// TIA Portal V20 export
// export: Created 2025-12-01T14:57:45.3823092Z, ExportSetting None, DisplayName Totally Integrated Automation Portal, DisplayVersion V20 Update 3, DisplayName TIA Portal Openness, DisplayVersion V20 Update 3, DisplayName TIA Portal Version Control Interface, DisplayVersion V20 Update 3, DisplayName STEP 7 Professional, DisplayVersion V20 Update 3, DisplayName STEP 7 Safety, DisplayVersion V20 Update 2, DisplayName WinCC Basic/Comfort/Advanced, DisplayVersion V20 Update 3, DisplayName WinCC Professional, DisplayVersion V20 Update 3, DisplayName WinCC Unified, DisplayVersion V20 Update 3
FUNCTION "FC818_Mensaje_BBDD_Routing_Llena" : Void   // FC818, LAD
{ S7_Optimized_Access := 'FALSE' }
// stored: AutoNumber false, SetENOAutomatically false
   VAR_INPUT
      Etiqueta : ULInt;
      Envio_JDT2 : Bool;
   END_VAR
   VAR_TEMP
      Guardar_AR1 : DWord;
      DBEventos : Word;   // Numero del DB de Eventos
      PunteroEventos : DWord;   // Puntero al DB de Eventos
      MaxBytes : UInt;
      NDB_Eventos_Emi : UInt;
      NumBytes : UInt;   // Numero de Bytes existentes en el DB de Eventos
      etiqueta_string : String;
      indice : Int;
      longitud : Int;
      posicion : Int;
      i : Int;
      codigo_string : String[20];
   END_VAR
BEGIN

REGION Network 1 (SCL)
   // buscamos hueco en el db donde vamos a escribir los eventos antes de empezar la conversión
   // 


   IF #Envio_JDT2    = true THEN
       REGION buscar en JDT2

           #posicion := -1;
           FOR #i := 0 TO 100 BY 1 DO
               #longitud := LEN("DB197_eventos_generados_routing_JDT2".evento[#i]);
               IF #longitud = 0 THEN
                   #posicion := #i;
                   EXIT;
               END_IF;
           END_FOR;

           // si no hay sitio para escribir salimos del bloque
           IF #posicion = -1 THEN
               RETURN;
           END_IF;
       END_REGION
       ;
   ELSE
       REGION buscar en JDT1

           #posicion := -1;
           FOR #i := 0 TO 100 BY 1 DO
               #longitud := LEN("DB198_eventos_generados_routing_JDT1".evento[#i]);
               IF #longitud = 0 THEN
                   #posicion := #i;
                   EXIT;
               END_IF;
           END_FOR;

           // si no hay sitio para escribir salimos del bloque
           IF #posicion = -1 THEN
               RETURN;
           END_IF;
       END_REGION
   END_IF;
END_REGION

REGION Network 2 (SCL): formatear el evento


   #codigo_string := DELETE(IN := (ULINT_TO_STRING(IN := #Etiqueta)), L := 1, P := 1);
   // concatenamos el mensaje 
   // 
   IF #Envio_JDT2= true THEN

       "DB197_eventos_generados_routing_JDT2".evento[#posicion] := CONCAT(IN1 := '{WARN[RUET]', IN2 := #codigo_string, IN3 := '[ERRO]BBDD[MOTI]FULL',  IN4 := "DB921_DATOS_FECHA_HORA".TIME_STAMP, IN5 := '}');

   ELSE
       "DB198_eventos_generados_routing_JDT1".evento[#posicion] :=CONCAT(IN1 := '{WARN[RUET]', IN2 := #codigo_string, IN3 := '[ERRO]BBDD[MOTI]FULL',  IN4 := "DB921_DATOS_FECHA_HORA".TIME_STAMP, IN5 := '}');

   END_IF;
END_REGION
END_FUNCTION
